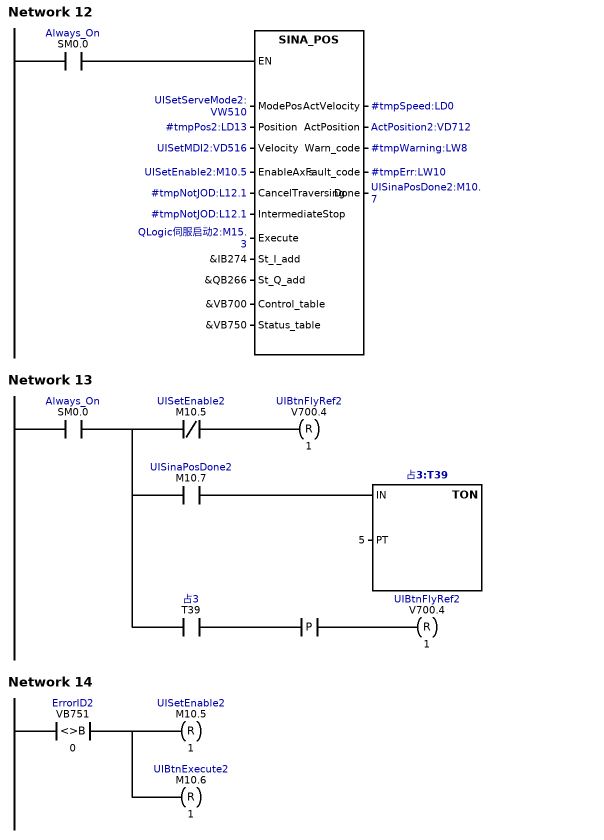
[picture p24: SBR9 networks 12-14]
Network 12
LD     Always_On:SM0.0
CALL   SINA_POS:SBR8, UISetServeMode2:VW510, #tmpPos2:LD13, UISetMDI2:VD516, UISetEnable2:M10.5, #tmpNotJOD:L12.1, #tmpNotJOD:L12.1, QLogic伺服启动2:M15.3, &IB274, &QB266, &VB700, &VB750, #tmpSpeed:LD0, ActPosition2:VD712, #tmpWarning:LW8, #tmpErr:LW10, UISinaPosDone2:M10.7
Network 13
LD     Always_On:SM0.0
LPS
AN     UISetEnable2:M10.5
R      UIBtnFlyRef2:V700.4, 1
LRD
A      UISinaPosDone2:M10.7
TON    占3:T39, 5
LPP
A      占3:T39
EU
R      UIBtnFlyRef2:V700.4, 1
Network 14
LDB<>  ErrorID2:VB751, 0
R      UISetEnable2:M10.5, 1
R      UIBtnExecute2:M10.6, 1
END_SUBROUTINE_BLOCK

// SBR10: protected block, not included

// SBR11: protected block, not included

// SBR12: protected block, not included
